TYPE ST_CHPDefaultParameters :
STRUCT
	fControllerAmplification : LREAL := 0.265;
	tControllerIntegralTime : TIME := T#15S;
	tTaskCycleTime	: TIME;
	tCtrlCycleTime	: TIME;
	aSetPointLimitsConstantPower : ARRAY[1..2] OF REAL := [0,100]; //setpoint limits for position mode
	aSetPointLimitsTemperature : ARRAY[1..2] OF REAL := [50,90]; //setpoint limits for temperature mode	
END_STRUCT
END_TYPE

(* stored: Version 1.1.0.1, ProductVersion 3.1.4024.10
   DUT ST_CHPDefaultParameters: Id {c6e10a81-b4a3-40b0-a4a6-e1b8857ffcd7} *)
